// TIA Portal V16 export
// export: Created 2020-03-29T17:41:57.7640743Z, ExportSetting None, DisplayName Totally Integrated Automation Portal, DisplayVersion V16 Update 1, DisplayName TIA Portal Version Control Interface, DisplayVersion V16, DisplayName TIA Portal Openness, DisplayVersion V16 Update 1, DisplayName SINAMICS Startdrive Advanced, DisplayVersion V16 Update 1, DisplayName SINAMICS Startdrive G130, G150, S120, S150, SINAMICS MV, S210, DisplayVersion V16 Update 1, DisplayName SINAMICS Startdrive G110M, G120, G120C, G120D, G120P, DisplayVersion V16 Update 1, DisplayName STEP 7 Professional, DisplayVersion V16 Update 1, DisplayName STEP 7 Safety, DisplayVersion V16, DisplayName WinCC Advanced, DisplayVersion V16 Update 1
FUNCTION_BLOCK "TemplateValve"   // FB2, LAD
TITLE = Sample valve template
{ S7_Optimized_Access := 'TRUE' }
// stored: MemoryReserve 100, SetENOAutomatically false
   VAR
      Valve_Instance { S7_SetPoint := 'True'} : "Valve";
   END_VAR
   VAR_TEMP
      Release : Bool;
      OpenValve : Bool;
      CloseValve : Bool;
   END_VAR
BEGIN

REGION Network 1: Release valve
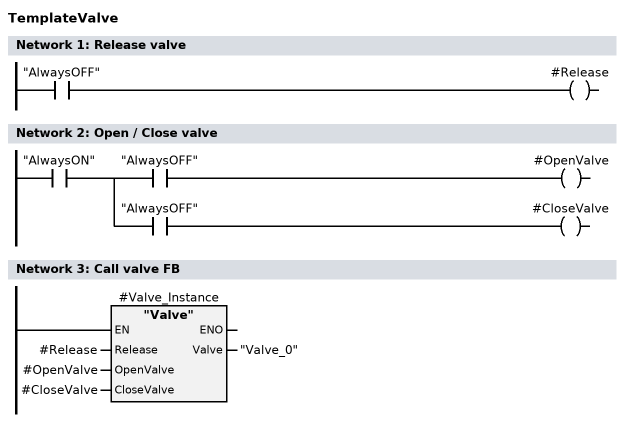
   RUNG wire#powerrail
      Contact( "AlwaysOFF" )
      Coil( #Release )
   END_RUNG
   // the same network as SCL:
   #Release := "AlwaysOFF";
END_REGION

REGION Network 2: Open / Close valve
   RUNG wire#powerrail
      Contact( "AlwaysON" )
      wire#w1
      Contact( "AlwaysOFF" )
      Coil( #OpenValve )
   END_RUNG
   RUNG wire#w1
      Contact( "AlwaysOFF" )
      Coil( #CloseValve )
   END_RUNG
   // the same network as SCL:
   #OpenValve := "AlwaysON" AND "AlwaysOFF";
   #CloseValve := "AlwaysON" AND "AlwaysOFF";
END_REGION

REGION Network 3: Call valve FB
   RUNG wire#powerrail
      #Valve_Instance(Release := #Release, OpenValve := #OpenValve, CloseValve := #CloseValve, Valve => "Valve_0")
   END_RUNG
   // the same network as SCL:
   #Valve_Instance(Release := #Release, OpenValve := #OpenValve, CloseValve := #CloseValve, Valve => "Valve_0");   // "Valve"
END_REGION
END_FUNCTION_BLOCK
